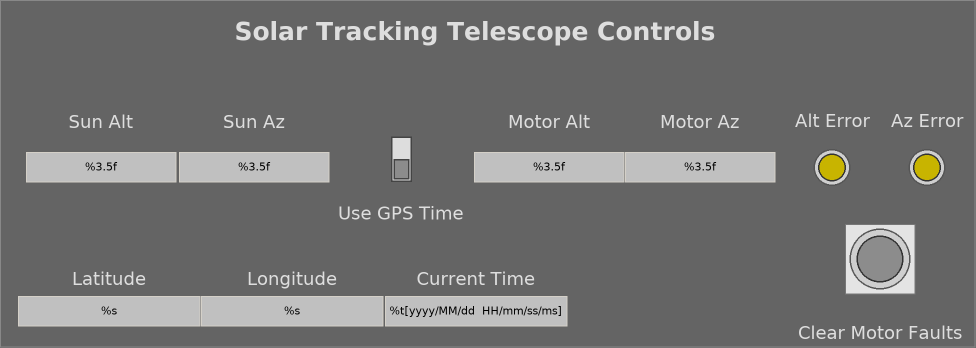
VISUALIZATION Visualization  // 976x348
    Label (217,5 516x52), "Solar Tracking Telescope Controls"
    Label (179,107 150x30), "Sun Az"
    Textfield (179,152 150x30), "%3.5f", text variable: MAIN.fSunAzimuth
    Label (26,107 150x30), "Sun Alt"
    Textfield (26,152 150x30), "%3.5f", text variable: MAIN.fSunAltitude
    Label (401,264 150x30), "Current Time"
    Textfield (385,296 182x30), "%t[yyyy/MM/dd HH/mm/ss/ms]", text variable: MAIN.currTime
    Textfield (625,152 150x30), "%3.5f", text variable: GVL.Az.NcToPlc.ActPos
    Label (625,107 150x30), "Motor Az"
    Textfield (474,152 150x30), "%3.5f", text variable: GVL.Alt.NcToPlc.ActPos
    Label (474,107 150x30), "Motor Alt"
    Label (34,264 150x30), "Latitude"
    Textfield (18,296 182x30), "%s", text variable: MAIN.fbSPA.fLatitude
    Label (217,264 150x30), "Longitude"
    Textfield (201,296 182x30), "%s", text variable: MAIN.fbSPA.fLongitude
    Group (785,106 190x83)
        Lamp1 (26,40 42x43), variable: MAIN.fbPositionMotors.Error_Alt, style: Lamp-Lamp1-Yellow
        Lamp1 (121,40 42x43), variable: MAIN.fbPositionMotors.Error_Az, style: Lamp-Lamp1-Yellow
        Label (0,0 95x30), "Alt Error"
        Label (95,0 95x30), "Az Error"
    PushSwitch (845,224 70x70), variable: MAIN.bResetMotors, behaviour: TOGGLE, style: Switch-PushSwitch-Gray
    Label (785,318 191x30), "Clear Motor Faults"
    DipSwitch (379,136 45x46), variable: MAIN.bUseGpsTime, behaviour: TOGGLE, style: Switch-DipSwitch-Gray
    Label (320,177 162x73), "Use GPS Time"
END_VISUALIZATION

(* stored: Version 1.1.0.1
   Visu Visualization: Id {345c444a-39b5-402c-a82f-0fda35e2ea9a} *)
